// TIA Portal V17 export
// export: Created 2024-08-26T21:10:50.6413411Z, ExportSetting WithDefaults, DisplayName Totally Integrated Automation Portal, DisplayVersion V17 Update 7, DisplayName TIA Portal Openness, DisplayVersion V17 Update 7, DisplayName TIA Portal Version Control Interface, DisplayVersion V17, DisplayName SINAMICS Startdrive Advanced, DisplayVersion V17 SP2, DisplayName SINAMICS Startdrive G110M, G120, G120C, G120D, G120P, G115D, DisplayVersion V17 SP2, DisplayName SINAMICS Startdrive G130, G150, S120, S150, SINAMICS MV, S210, DisplayVersion V17 SP2, DisplayName STEP 7 Professional, DisplayVersion V17 Update 7, DisplayName STEP 7 Safety, DisplayVersion V17 Update 6, DisplayName WinCC Advanced / Unified PC, DisplayVersion V17 Update 7
DATA_BLOCK "DB_HMI"   // DB7
{ S7_Optimized_Access := 'TRUE' }
VERSION : 0.1
// stored: AutoNumber true, DBAccessibleFromOPCUA true, DBAccessibleFromWebserver true, IsOnlyStoredInLoadMemory false, IsRetainMemResEnabled false, IsWriteProtectedInAS false, MemoryReserve 100
   VAR
      modeButton : Bool := FALSE;
      mode : Int := 2;
      model : Array[0..32] of Bool;
      recipeStep : Int := 3;
      "a" : DInt := -2_146_096_376;
      "b" : DInt := 4197;
      mascA : DInt := 134_221_952;
      mascB : DInt := 0;
      recipeStepTime : Int := 500;
      recipeStepSubstract : Bool := FALSE;
      recipeStepAdd : Bool := FALSE;
      recipeLastStep : Int := 3;
      updateStep : Bool := FALSE;
      moveToCurrentStep : Bool := FALSE;
      recordA1 : Bool := FALSE;
      readA1 : Bool := FALSE;
      recordA2 : Bool := FALSE;
      readA2 : Bool := FALSE;
      recordB1 : Bool := FALSE;
      readB1 : Bool := FALSE;
      recordB2 : Bool := FALSE;
      readB2 : Bool := FALSE;
      recordAnalog : Bool := FALSE;
      readAnalog : Bool := FALSE;
      recipeStepQuantity : Int := 8;
      eraseStep : Bool := FALSE;
      insertStep : Bool := FALSE;
      copyStep : Bool := FALSE;
      copySequence : Bool := FALSE;
      copySequenceStep : Bool := FALSE;
      baseStep : Int := 7;
      destinationStep : Int := 8;
      baseModel : Int := 3;
      destinationModel : Int := 6;
      baseModelStep : Int := 0;
      modelDestinationStep : Int := 0;
      baseModelStep_1 : Int := 2;
      modelDestinationStep_1 : Int := 3;
      operatorTextIndicator : String := ' ';
      enableStationAir : Bool := FALSE;
      enableAirHmiPermission : Bool := FALSE;
      insertAlarmKey : Bool := FALSE;
      enableStationVisualizationButton : Bool := FALSE;
      enableStationHideAlarmButton : Bool := FALSE;
      alarmAckmowledge : Bool := FALSE;
      home : Bool := FALSE;
      advancePercentage : Real := 0.0;
      administratorAlarmButton : Bool := FALSE;
      activateLamp : Bool := TRUE;
      activateFan : Bool := TRUE;
   END_VAR
   VAR RETAIN
      cicles : Int := 285;
      production1 : Int := 247;
      production2 : Int := 56;
      production3 : Int := 0;
   END_VAR
   VAR
      productionRestart1 : Bool := FALSE;
      productionRestart2 : Bool := FALSE;
      productionRestart3 : Bool := FALSE;
      ciclesRestart : Bool := FALSE;
      manualPrint : Bool := FALSE;
      BLOQUEO : Bool := TRUE;
      manualModeNecessary : Bool := FALSE;
      modelChange : Bool := FALSE;
      alarmManualButton : Bool := FALSE;
      user : String := 'Administrator';
      pass : String := 'PASSWORD';
   END_VAR
BEGIN
   model[0..32] := FALSE;
END_DATA_BLOCK
